// TIA Portal V20 export
DATA_BLOCK "DB_Alarm"   // DB15
// stored: Access Published, MemoryReserve 100, Namespace LineD1
   VAR
      "word" : Struct
         Line : Struct
            D1 : Struct
               Conveyor : Array[_.minD1.._.maxD1] of Word;
            END_STRUCT;
         END_STRUCT;
      END_STRUCT;
   END_VAR
BEGIN
END_DATA_BLOCK
